//{attribute 'qualified_only'}
{attribute 'strict'}
TYPE E_Command :
(
	 eReady, 
	 eFwd, 
	 eRev,
	 eResetInv  
	 
); // domyślna inicjalizacja wszystkich E_ATVCommand Variables na WORD
END_TYPE

(* stored: Version 1.1.0.1, ProductVersion 3.1.4024.12
   DUT E_Command: Id {d50d8559-d507-4ce1-81cc-42f496ab1cf0} *)
